FUNCTION Convert_SINT_TO_LREAL : Hresult
VAR_INPUT
	in : SINT;
	out : REFERENCE TO LREAL;
END_VAR
VAR
	converted : LREAL;
END_VAR
VAR CONSTANT
	INCOMPATIBLE : HRESULT := 16#9811070E;
END_VAR

converted := SINT_TO_LREAL(in);

IF (LREAL_TO_SINT(converted) <> in) THEN
	Convert_SINT_TO_LREAL := INCOMPATIBLE;
	RETURN;
END_IF

out := converted;

END_FUNCTION

(* stored: Version 1.1.0.1, ProductVersion 3.1.4024.12
   POU Convert_SINT_TO_LREAL: Id {366ebcc7-1f6a-4a9b-a216-b264b81d752a}, SpecialFunc None *)
